TYPE S_Setting :
STRUCT
	Code: STRING[4];
	Description: STRING[256];
	Value: REAL;
	Unit: STRING[10];
END_STRUCT
END_TYPE

(* stored: Version 1.1.0.1, ProductVersion 3.1.4024.0
   DUT S_Setting: Id {132016bc-b80f-4dbb-bf4d-2cc0ec72e2f4} *)
